// SIMATIC S7-200 SMART project (STEP 7-Micro/WIN SMART), CPU SR20

SYMBOL_TABLE System Symbols
Always_On        SM0.0    // Always ON
END_SYMBOL_TABLE

ORGANIZATION_BLOCK MAIN:OB1
TITLE=Program Comments
BEGIN
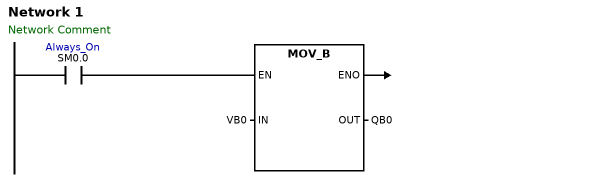
Network 1
// Network Comment
LD     Always_On:SM0.0
MOVB   VB0, QB0
END_ORGANIZATION_BLOCK

DATA_BLOCK_TAB Page_1
BEGIN
//DATA PAGE COMMENTS
//Press F1 for help and example data page
VB0      5
END_DATA_BLOCK_TAB
